// TIA Portal V18 export
DATA_BLOCK "pressure"   // DB71
{ S7_Optimized_Access := 'TRUE' }
VERSION : 0.1
// stored: AutoNumber true, DBAccessibleFromOPCUA true, IsOnlyStoredInLoadMemory false, IsRetainMemResEnabled false, IsWriteProtectedInAS false, MemoryReserve 100
   VAR RETAIN
      "A" : Struct
         "pressure at 20mA" : Real := 160.0;
         "Maximum Pressure user" : Real := 10.0;
         "maximum pressure Admin" : Real := 10.0;
         "minimum Pressure" : Real := 1.5;
      END_STRUCT;
      "B" : Struct
         "pressure at 20mA" : Real := 160.0;
         "Maximum Pressure user" : Real := 10.0;
         "maximum pressure Admin" : Real := 10.0;
         "minimum Pressure" : Real := 1.5;
      END_STRUCT;
   END_VAR
   VAR
      "Control A" : Struct
         "Over pressure occured" : Bool := FALSE;
         "under pressure Occured" : Bool := FALSE;
      END_STRUCT;
      "Control B" : Struct
         "Over pressure occured" : Bool := FALSE;
         "under pressure Occured" : Bool := FALSE;
      END_STRUCT;
      "pump A Inlet" : Real := 1.50463;
      "pump B Inlet" : Real := 1.545139;
      "pump A Outlet" : Real := 0.1808449;
      "pump B Outlet" : Real := 0.1139323;
      "Vessel A1 mbar" : DInt := 0;
      "Vessel A2 mbar" : DInt := 0;
      "Vessel B2 mbar" : DInt := 0;
      "Vessel B1 mbar" : DInt := 0;
   END_VAR
   VAR RETAIN
      "Over pressure Delay time user" : DInt := 1000;
      "over pressure delay time admin" : DInt := 10000;
      "under pressure delay time" : DInt := 1000;
      "Vaccum  sensor range" : Struct
         A1mbar : DInt := 9000;
         A2mbar : DInt := 9000;
         B1mbar : DInt := 9000;
         B2mbar : DInt := 9000;
         A1bar : Real := 9.0;
         A2bar : Real := 9.0;
         B1bar : Real := 9.0;
         B2bar : Real := 0.0;
      END_STRUCT;
   END_VAR
   VAR
      "vessel A1 bar" : Real := 0.0;
      "vessel A2 bar" : Real := 0.0;
      "vessel B1 bar" : Real := 0.0;
      "vessel B2 bar" : Real := 0.0;
      Misc : Struct
         "Pump A normx valueIN" : Real := 0.009403936;
         "Pump B normx valueIN" : Real := 0.009657118;
         "Pump A Scalx valueIN" : Real := 1.50463;
         "Pump B Scalx valueIN" : Real := 1.545139;
         "Pump A normx valueOUT" : Real := 0.007233796;
         "Pump B normx valueOUT" : Real := 0.004557292;
         "Pump A Scalx valueOUT" : Real := 0.1808449;
         "Pump B Scalx valueOUT" : Real := 0.1139323;
         "normx Tank A1" : Real := 0.0;
         "normx Tank A2" : Real := 0.0;
         "normx Tank B1" : Real := 0.0;
         "normx Tank B2" : Real := 0.0;
         "scalx Tank A1" : Real := 0.0;
         "scalx Tank A2" : Real := 0.0;
         "scalx Tank B1" : Real := 0.0;
         "scalx Tank B2" : Real := 0.0;
      END_STRUCT;
      "Control Vessel A1" : Struct
         "under pressure" : Bool := FALSE;
         "Over pressure open release valve" : Bool := FALSE;
      END_STRUCT;
      "Control Vessel A2" : Struct
         "under pressure" : Bool := FALSE;
         "Over pressure open release valve" : Bool := FALSE;
      END_STRUCT;
      "Control Vessel B1" : Struct
         "under pressure" : Bool := FALSE;
         "Over pressure open release valve" : Bool := FALSE;
      END_STRUCT;
      "Control Vessel B2" : Struct
         "under pressure" : Bool := FALSE;
         "Over pressure open release valve" : Bool := FALSE;
      END_STRUCT;
   END_VAR
   VAR RETAIN
      A_Outlet : Struct
         "pressure at 20mA" : Real := 25.0;
         "Maximum Pressure user" : Real := 20.0;
         "maximum pressure Admin" : Real := 20.0;
         "minimum Pressure" : Real := 1.0;
      END_STRUCT;
      B_Outlet : Struct
         "pressure at 20mA" : Real := 25.0;
         "Maximum Pressure user" : Real := 20.0;
         "maximum pressure Admin" : Real := 20.0;
         "minimum Pressure" : Real := 1.0;
      END_STRUCT;
   END_VAR
   VAR
      "Control A_Outlet" : Struct
         "Over pressure occured" : Bool := FALSE;
         "under pressure Occured" : Bool := FALSE;
      END_STRUCT;
      "Control B_Outlet" : Struct
         "Over pressure occured" : Bool := FALSE;
         "under pressure Occured" : Bool := FALSE;
      END_STRUCT;
   END_VAR
   VAR RETAIN
      Outlet_PT_ENABLE : Bool := TRUE;
   END_VAR
BEGIN
END_DATA_BLOCK
